TYPE ST_RAA_6_0_CommandArgs :
STRUCT
	Key			: STRING(SIS_6_0.RAA_COMMAND_ARGS_KEY_STRINGLENGTH); // Key
	Value		: STRING(SIS_6_0.RAA_COMMAND_ARGS_VALUE_STRINGLENGTH); // Value
END_STRUCT
END_TYPE

(* stored: Version 1.1.0.1, ProductVersion 3.1.4022.12
   DUT ST_RAA_6_0_CommandArgs: Id {9dc92cf6-c99b-43b7-8006-9f11c2f94a4f} *)
